Fanuc KAREL source: ka00090.KL

-- PROVISIONAL review KL for V1013-1; original PC SHA256 d2ccb8fe028063a2943ae8785c303cce023c71edc0d69a34fc2f24129d623caf
-- Incomplete behavior may be omitted. Consult companion uncertainty JSON. Do not deploy.
PROGRAM KA00090
%NOLOCKGROUP
-- UNRESOLVED_DECL SRC type=000199
-- UNRESOLVED_DECL DST type=000102
BEGIN
  -- UNRESOLVED_PC offsets 5-25; opcodes 49,7E,4A
  -- UNRESOLVED_PC offsets 30-34; opcodes 7F
END KA00090
